RoboDK station: Assembly cell.rdk

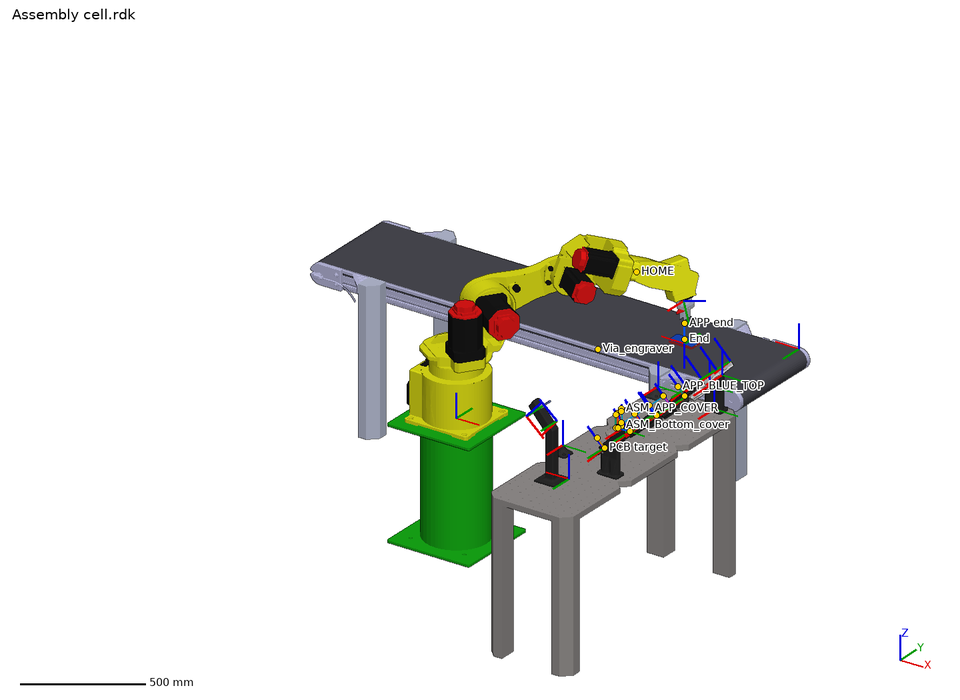
[picture v0: the station drawn from its stored meshes, robots at their saved joint values, targets as dots, program paths as lines]
Station Assembly cell. Poses are relative to the parent item; angles as X-Y-Z fixed-axis rotations.
  - program Assemble Blue phone (11 instructions, listed below)
  - program Assemble Red phone (11 instructions, listed below)
  - folder Frames
    - frame Conveyor Belt Base at (960, 1000, 175) mm, rotated rx 0 ry 0 rz -180 deg
      - robot Conveyor Belt: 1 axes
          modified DH rows (alpha deg, a mm, theta deg, d mm): 0, 0, 0, 0 linear
          base shift (0, 0, 0) mm, rotated rx 0 ry 90 rz 0 deg
          joint limits [-500000] to [500000]; home [0]; saved at [0]
      - frame End distination at (400, 220, 0) mm, rotated rx 180 ry 0 rz 0 deg
        - target End (Cartesian target) at (0, 0, -17.7) mm; joints [55.844, 86.591, -24.189, 14.611, -58.106, -62.758] of M-6IB
        - target APP end  (Cartesian target) at (0, 0, -90) mm; joints [-32.781, 53.881, -40.537, 165.227, 58.581, -48.481] of M-6IB
      - object Ben til Anton samleba at (311, -3, 0) mm, rotated rx -90 ry 0 rz 0 deg, size 80 x 676 x 80 mm, geometry from nd.STEP
      - object Ben til Anton samleba at (1774, -3, 0) mm, rotated rx -90 ry 0 rz -90 deg, size 80 x 676 x 80 mm, geometry from nd.STEP
      - object Ben til Anton samleba at (311, 443, 0) mm, rotated rx -90 ry 0 rz 90 deg, size 80 x 676 x 80 mm, geometry from nd.STEP
      - object Ben til Anton samleba at (1773, 443, 0) mm, rotated rx -90 ry 0 rz 180 deg, size 80 x 676 x 80 mm, geometry from nd.STEP
    - frame M-6IB Base at (0, 0, 0) mm
      - robot M-6IB: 6 axes
          modified DH rows (alpha deg, a mm, theta deg, d mm): 0, 0, 0, 450; -90, 150, -90, 0; 0, 360, 0, 0; -90, 100, 0, 430; 90, 0, 0, 0; -90, 0, 180, 100
          joint limits [-170, -90, -80, -190, -140, -360] to [170, 160, 80, 190, 140, 360]; home [0, 0, 0, 0, 0, 0]; saved at [55.844, 79.928, -20.148, 14.035, -62.022, -61.604]
        - tool TCP_Cover, TCP at (20.4, 0, 95.1) mm, rotated rx 0 ry 15 rz 0 deg
        - tool TCP_DrawingTool(slet mig), TCP at (25.5, 0, 114.13) mm, rotated rx 0 ry 15 rz 0 deg
        - tool TCP_DrawingToolCorner, TCP at (8.96, -4.5, 118.56) mm, rotated rx 180 ry 15 rz 0 deg
        - tool TCP_FUSE, TCP at (19.7, 0, 92.49) mm, rotated rx 0 ry 15 rz 0 deg
        - frame Gripper at (0, 0, 0) mm, rotated rx 90 ry 0 rz -90 deg
          - robot Gripper: 1 axes
              joint limits [0] to [16]; home [0]; saved at [5]
          - target Close (Cartesian target) at (0, 0, 150) mm; joints [0.01] of Gripper
          - target Open (Cartesian target) at (0, 0, 150) mm; joints [5] of Gripper
        - tool TCP_PCB, TCP at (-16.6, 0, 115.3) mm, rotated rx 15 ry 0 rz 90 deg
      - frame Worktable at (700, 400, 175) mm, rotated rx 0 ry 0 rz -90 deg
        - object WorkTable at (20, 20, 0) mm, rotated rx 90 ry 0 rz 0 deg, size 1200 x 700 x 400 mm, geometry from WorkTable.3sections.STEP
        - frame Assembler at (400, 100, 0) mm
          - object Assembler.fixture at (-90, -50, 4) mm, rotated rx -90 ry 0 rz -90 deg, size 70 x 14 x 180 mm, geometry from Assembler.fixture.STEP
          - target ASM_APP_COVER (Cartesian target) at (0, 0, 90) mm, rotated rx -180 ry 0 rz 0 deg; joints [-2.519, 35.979, -52.892, -23.6, -40.23, 111.053] of M-6IB
          - target ASM_APP_FUSE1 (Cartesian target) at (26.19, 0, 80) mm, rotated rx 180 ry 0 rz -90 deg; joints [-2.241, 33.623, -56.565, -1.832, -18.455, 3.903] of M-6IB
          - target ASM_APP_FUSE2 (Cartesian target) at (39.25, 0, 80) mm, rotated rx 180 ry 0 rz -90 deg; joints [-3.357, 33.698, -56.518, -2.734, -18.526, 5.835] of M-6IB
          - target ASM_APP_PCB (Cartesian target) at (0, 0, 80) mm, rotated rx 180 ry 0 rz -180 deg; joints [2.519, 37.294, -54.217, 24.249, -39.018, -111.896] of M-6IB
          - target ASM_Bottom_cover (Cartesian target) at (0, 0, 17) mm, rotated rx 180 ry 0 rz 0 deg; joints [-2.519, 44.305, -60.421, -27.98, -33.444, -243.485] of M-6IB
          - target ASM_FUSE1 (Cartesian target) at (26.19, 0, 19.5) mm, rotated rx 180 ry 0 rz -90 deg; joints [-2.241, 40.726, -62.911, -2.764, -12.114, 4.868] of M-6IB
          - target ASM_FUSE2 (Cartesian target) at (39.25, 0, 19.5) mm, rotated rx 180 ry 0 rz -90 deg; joints [-3.357, 40.792, -62.856, -4.112, -12.199, 7.262] of M-6IB
          - target ASM_GRAB_PHONE (Cartesian target) at (0, 0, 23.7) mm, rotated rx -180 ry 0 rz 0 deg; joints [-2.519, 43.211, -59.538, -27.369, -34.225, 115.779] of M-6IB
          - target ASM_PCB (Cartesian target) at (0, 0, 14.5) mm, rotated rx 180 ry 0 rz 180 deg; joints [0, 25.65, -72.841, 0, -2.159, 0] of M-6IB
          - target ASM_TOP_cover (Cartesian target) at (0, 0, 28.7) mm, rotated rx 180 ry 0 rz 0 deg; joints [-2.519, 42.635, -59.062, -27.052, -34.649, 115.394] of M-6IB
          - object Assembler.fixture at (-90, -50, 4) mm, rotated rx -90 ry 0 rz -90 deg, size 70 x 14 x 180 mm, geometry from Assembler.fixture.STEP
          - target HOME (Cartesian target) at (0, 75.1, 714.6) mm, rotated rx -180 ry 75 rz -90 deg; joints [0, 0, 0, 0, 0, 0] of M-6IB
          - object Sikring at (-790, -279.25, 13.5) mm, rotated rx 0 ry -45 rz -90 deg, size 5 x 20 x 5 mm, geometry from Sikring.STEP
          - object Sikring at (-790, -266.19, 13.5) mm, rotated rx 0 ry -45 rz -90 deg, size 5 x 20 x 5 mm, geometry from Sikring.STEP
          - object PCB at (-780, -245.3, 6.2) mm, rotated rx -90 ry 0 rz 0 deg, size 55 x 11.2 x 106.7 mm, geometry from PCB.STEP
          - object BundRed at (-780, -240, 11) mm, rotated rx 0 ry 0 rz -90 deg, size 60 x 13 x 114 mm, geometry from BundRed.STEP
          - object TopBlue at (-780, -240, 17.7) mm, rotated rx 0 ry 0 rz -90 deg, size 60 x 11.7 x 114 mm, geometry from TopBlue.STEP
        - frame Calibration tip 2 at (720, 40, 40) mm
          - object Calibration tip2 - Table at (0, 0, -40) mm, rotated rx 90 ry 0 rz 0 deg, size 64 x 40 x 64 mm, geometry from Calibration tip - Table.STEP
        - frame Engraving tool at (890, 190, 0) mm, rotated rx 0 ry 0 rz -90 deg
          - frame Pencil at (171.86, 50, 249.32) mm, rotated rx 0 ry 41.29 rz -180 deg
            - target Via_engraver (Cartesian target) at (-59.9, 461.47, 104.18) mm, rotated rx -165.52 ry -18.84 rz -114.89 deg; joints [-18.02, 30.15, -78.63, -152.85, -139.18, 114.67] of M-6IB
          - frame Pencil corner(slet mig) at (31.87, 41, 263.19) mm, rotated rx 0 ry 48.71 rz 0 deg
          - object Engraving Tool at (0, 0, 0) mm, rotated rx -90 ry 0 rz 0 deg, size 171.9 x 351.3 x 100 mm, geometry from Pencil.assembly.STEP
        - frame Left Pillar at (40, 300, 0) mm
          - frame Rod lower at (-11.02, -32.53, 91.11) mm
            - object Rod at (0, 0, 0) mm, size 8 x 742 x 8 mm, geometry from Rod.STEP
            - frame Assembly blue bottom cover 1 at (250, 137.68, 167.7) mm, rotated rx 0 ry 45 rz -90 deg
              - frame target_blue_bottom_cover at (280, 35.13, -4.5) mm
                - target Blue_bottom (Cartesian target) at (0, 0, 0) mm, rotated rx 180 ry 0 rz 0 deg; joints [7.51, 44.296, -67.681, -10.607, 37.945, 4.63] of M-6IB
                - target APP_Blue_bottom (Cartesian target) at (0, 0, 50) mm, rotated rx 180 ry 0 rz 0 deg; joints [7.935, 36.225, -67.101, -11.351, 37.406, 5.073] of M-6IB
                - object BundBlue at (0, 0, 0) mm, size 60 x 13 x 114 mm, geometry from BundBlue.STEP
              - object Top cover fixture at (0, 0, 0) mm, size 70.2 x 39.6 x 342 mm, geometry from Top cover fixture.STEP
              - object FixtureBlack at (0, 0, 1.25) mm, rotated rx 0 ry 0 rz 180 deg, size 342 x 70.2 x 41.2 mm, geometry from FixtureBlack.STEP
            - frame Assembly blue top cover 1 at (50, 137.68, 167.7) mm, rotated rx 0 ry 45 rz -90 deg
              - frame target_blue_top_cover at (280, 35.12, -4.5) mm
                - target BLUE_TOP (Cartesian target) at (0, 0, 5) mm, rotated rx 180 ry 0 rz 0 deg; joints [23.805, 48.879, -62.525, -36.506, 35.985, 18.478] of M-6IB
                - target APP_BLUE_TOP (Cartesian target) at (0, 0, 50) mm, rotated rx 180 ry 0 rz 0 deg; joints [24.889, 42.011, -62.308, -38.195, 36.117, 19.379] of M-6IB
              - object Top cover fixture at (0, 0, 0) mm, size 70.2 x 39.6 x 342 mm, geometry from Top cover fixture.STEP
            - frame Assembly red bottom cover 2 at (350, 137.68, 167.7) mm, rotated rx 0 ry 45 rz -90 deg
              - frame target_red_bottom_cover at (280, 35.12, -4.5) mm
                - target Red_bottom (Cartesian target) at (0, 0, 0) mm, rotated rx 180 ry 0 rz 0 deg; joints [-1.236, 44.216, -68.191, 181.732, -38.198, -180.743] of M-6IB
                - target APP_Red_bottom (Cartesian target) at (0, 0, 50) mm, rotated rx 180 ry 0 rz 0 deg; joints [-1.307, 36.105, -67.625, 181.854, -37.633, -180.815] of M-6IB
              - object FixtureBlack at (0, 0, 1.25) mm, rotated rx 0 ry 0 rz 180 deg, size 342 x 70.2 x 41.2 mm, geometry from FixtureBlack.STEP
            - frame Assembly red top cover 2 at (150, 137.68, 167.7) mm, rotated rx 0 ry 45 rz -90 deg
              - object Top cover fixture at (0, 0, 0) mm, size 70.2 x 39.6 x 342 mm, geometry from Top cover fixture.STEP
              - frame target_red_top_cover at (280, 35.12, -4.5) mm
                - target Red_top (Cartesian target) at (0, 0, 5) mm, rotated rx 180 ry 0 rz 0 deg; joints [16.006, 45.457, -65.78, -23.315, 37.109, 10.806] of M-6IB
                - target APP_Red_top (Cartesian target) at (0, 0, 50) mm, rotated rx 180 ry 0 rz 0 deg; joints [16.787, 38.357, -65.346, -24.653, 36.843, 11.591] of M-6IB
                - object TopRed at (0, 0, 0) mm, size 60 x 11.7 x 114 mm, geometry from TopRed.STEP
              - object Top cover fixture at (0, 0, 0) mm, size 70.2 x 39.6 x 342 mm, geometry from Top cover fixture.STEP
            - frame Fuses fixture at (500, 83.09, 94.4) mm, rotated rx 0 ry 45 rz -90 deg
              - frame fuse target at (154.59, 6.25, 7) mm
                - target Fuse target (Cartesian target) at (0, 0, 0) mm, rotated rx 135 ry 0 rz -90 deg; joints [-10.843, 50.524, -86.333, -184.166, -86.343, 90.266] of M-6IB
                - target APP_Target_fuse (Cartesian target) at (40, 0, 40) mm, rotated rx 180 ry 0 rz -90 deg; joints [-9.229, 37.854, -63.685, -23.305, 21.644, -61.596] of M-6IB
                - object Sikring at (0, -10, 0) mm, size 5 x 20 x 5 mm, geometry from Sikring.STEP
                - object Sikring at (0, -10, 0) mm, size 5 x 20 x 5 mm, geometry from Sikring.STEP
              - object FuseFixture at (0, 0, 0) mm, size 28.5 x 33.2 x 160 mm, geometry from FuseFixture.STEP
            - frame PCB fixture at (600, 90.16, 101.47) mm, rotated rx 0 ry 45 rz -90 deg
              - frame pcb target at (187.5, 64.5, 6.5) mm
                - target PCB target (Cartesian target) at (0, -5.3, 0) mm, rotated rx 180 ry 0 rz -90 deg; joints [-28.731, 41.343, -74.438, -145.13, -46.732, -190.202] of M-6IB
                - target APP_PCB (Cartesian target) at (0, -5.3, 50) mm, rotated rx 180 ry 0 rz -90 deg; joints [0, 0, 0, 0, 0, 0] of M-6IB
              - object PCB fixture at (0, 0, 0) mm, rotated rx 90 ry 0 rz 90 deg, size 118 x 39.5 x 220 mm, geometry from PCB fixture.STEP
          - frame Rod upper at (-11.02, 31.11, 154.75) mm
            - object Rod at (0, 0, 0) mm, size 8 x 742 x 8 mm, geometry from Rod.STEP
          - object Pillar at (0, 0, 0) mm, rotated rx 90 ry 0 rz 0 deg, size 60 x 165 x 100 mm, geometry from Søjle.STEP
        - frame Right Pillar at (760, 300, 0) mm
          - object Pillar at (0, 0, 0) mm, rotated rx 90 ry 0 rz 0 deg, size 60 x 165 x 100 mm, geometry from Søjle.STEP
        - frame Calibration tip 1 at (80, 40, 40) mm
          - object Calibration tip - Table at (0, 0, -40) mm, rotated rx 90 ry 0 rz 0 deg, size 64 x 40 x 64 mm, geometry from Calibration tip - Table.STEP
  - folder Programs
    - folder Attach Programs
      - program Attach_Bottom_Cover_Blue (8 instructions, listed below)
      - program Attach_Bottom_Cover_Red (8 instructions, listed below)
      - program Attach_Top_Cover_Blue (8 instructions, listed below)
      - program Attach_Top_Cover_Red (8 instructions, listed below)
      - program Attach_PCB (8 instructions, listed below)
      - program Attach_phone (10 instructions, listed below)
      - program Attach_Fuse (8 instructions, listed below)
    - folder Detach Programs
      - program Detach_Fuse1 (6 instructions, listed below)
      - program Detach_Fuse2 (6 instructions, listed below)
      - program Detach_PCB (7 instructions, listed below)
      - program Detach_Bottom (6 instructions, listed below)
      - program Detach_Top (5 instructions, listed below)
    - folder Misc
      - frame Robotbase_frame at (0, 0, -525) mm
        - object RobotBase at (-200, -200, 0) mm, rotated rx 90 ry 0 rz 0 deg, size 400 x 525 x 400 mm, geometry from RobotBase.STEP
      - program Open gripper (4 instructions, listed below)
      - program Close gripper (1 instructions, listed below)
      - Python program Generate G-Code (listed below)
      - Python program Import G-Code (listed below)
      - program Final step (6 instructions, listed below)
    - program Reset 2 (1 instructions, listed below)
    - folder Programs for Test
      - program Red phone assembly test (2 instructions, listed below)
      - program Blue phone assembly test (2 instructions, listed below)
  - Python program Assemble red phone (listed below)
  - program Reset (2 instructions, listed below)
  - Python program Assemble blue phone (listed below)
  - program AssembleInterior (6 instructions, listed below)
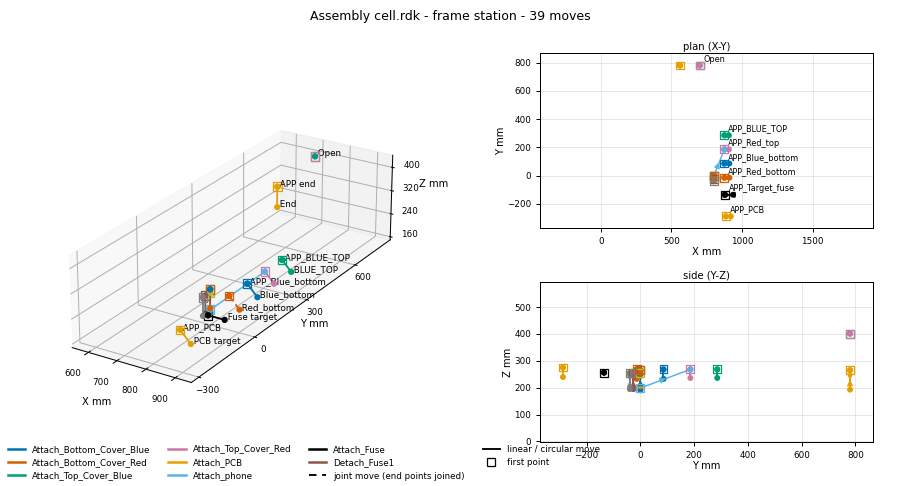
[picture p0: tool path of Assembly cell.rdk in frame station, 39 of 39 moves have a stored position in this frame; points joined in program order, loops and branches not executed]

--- program Assemble Blue phone (robot M-6IB) ---
  Call Attach_Bottom_Cover_Blue
  Call Detach_Bottom
  Call Attach_PCB
  Call Detach_PCB
  Call Attach_Fuse
  Call Detach_Fuse1
  Call Attach_Fuse
  Call Detach_Fuse2
  Call Attach_Top_Cover_Blue
  Call Detach_Top
  Call Final step

--- program Assemble Red phone (robot M-6IB) ---
  Call Attach_Bottom_Cover_Red
  Call Detach_Bottom
  Call Attach_PCB
  Call Detach_PCB
  Call Attach_Fuse
  Call Detach_Fuse1
  Call Attach_Fuse
  Call Detach_Fuse2
  Call Attach_Top_Cover_Red
  Call Detach_Top
  Call Final step

--- program Attach_Bottom_Cover_Blue (robot M-6IB) ---
  Set Tool: TCP_Cover
  Set Ref.: target_blue_bottom_cover
  Call Open
  MoveJ (APP_Blue_bottom)
  MoveL (Blue_bottom)
  Attach to TCP_PCB
  Call Close gripper
  MoveL (APP_Blue_bottom)

--- program Attach_Bottom_Cover_Red (robot M-6IB) ---
  Set Tool: TCP_Cover
  Set Ref.: target_red_bottom_cover
  Call Open
  MoveJ (APP_Red_bottom)
  MoveJ (Red_bottom)
  Attach to TCP_PCB
  Call Close gripper
  MoveJ (APP_Red_bottom)

--- program Attach_Top_Cover_Blue (robot M-6IB) ---
  Set Tool: TCP_Cover
  Set Ref.: target_blue_top_cover
  Call Open
  MoveJ (APP_BLUE_TOP)
  MoveL (BLUE_TOP)
  Attach to TCP_PCB
  Call Close gripper
  MoveL (APP_BLUE_TOP)

--- program Attach_Top_Cover_Red (robot M-6IB) ---
  Set Tool: TCP_Cover
  Set Ref.: target_red_top_cover
  Call Open
  MoveJ (APP_Red_top)
  MoveL (Red_top)
  Attach to TCP_PCB
  Call Close gripper
  MoveL (APP_Red_top)

--- program Attach_PCB (robot M-6IB) ---
  Set Tool: TCP_PCB
  Set Ref.: pcb target
  Call Open
  MoveJ (APP_PCB)
  MoveL (PCB target)
  Attach to TCP_PCB
  Call Close gripper
  MoveL (APP_PCB)

--- program Attach_phone (robot M-6IB) ---
  Set Tool: TCP_Cover
  Set Ref.: Assembler
  MoveL (ASM_GRAB_PHONE)
  Call Close gripper
  Attach to TCP_Cover
  Attach to TCP_Cover
  Attach to TCP_Cover
  Attach to TCP_Cover
  Attach to TCP_Cover
  MoveL (APP_Red_top)

--- program Attach_Fuse (robot M-6IB) ---
  Set Tool: TCP_FUSE
  Set Ref.: fuse target
  Call Open
  MoveJ (APP_Target_fuse)
  MoveL (Fuse target)
  Attach to TCP_PCB
  Call Close gripper
  MoveL (APP_Target_fuse)

--- program Detach_Fuse1 (robot M-6IB) ---
  Set Ref.: Assembler
  Set Tool: TCP_FUSE
  MoveJ (ASM_APP_FUSE1)
  MoveL (ASM_FUSE1)
  Call Open gripper
  MoveL (ASM_APP_FUSE1)

--- program Detach_Fuse2 (robot M-6IB) ---
  Set Ref.: Assembler
  Set Tool: TCP_FUSE
  MoveJ (ASM_APP_FUSE2)
  MoveL (ASM_FUSE2)
  Call Open gripper
  MoveL (ASM_APP_FUSE2)

--- program Detach_PCB (robot M-6IB) ---
  Set Ref.: Assembler
  Set Tool: TCP_PCB
  MoveJ (ASM_APP_PCB)
  MoveL (ASM_PCB)
  Call Open gripper
  Replace PCB
  MoveL (ASM_APP_PCB)

--- program Detach_Bottom (robot M-6IB) ---
  Set Ref.: Assembler
  Set Tool: TCP_Cover
  MoveJ (ASM_APP_COVER)
  MoveL (ASM_Bottom_cover)
  Call Open gripper
  MoveL (ASM_APP_COVER)

--- program Detach_Top (robot M-6IB) ---
  Set Ref.: Assembler
  Set Tool: TCP_Cover
  MoveJ (ASM_APP_COVER)
  MoveL (ASM_TOP_cover)
  Call Open gripper

--- program Open gripper (robot Gripper) ---
  MoveJ (Open)
  Detach from TCP_Cover
  Detach from TCP_PCB
  Detach from TCP_FUSE

--- program Close gripper (robot Gripper) ---
  MoveJ (Close)

--- Python program Generate G-Code ---
# Typo created by Adrien Rosselet

from os import path               # Operating System API
from robolink import *    # RoboDK API
from robodk import *      # Robot toolbox
#import time
import sys                # System specific
#Connect to RoboDK
RDK = Robolink()

#If no input the text equals ROBOT.
text = 'ROBOT'
#Use function call argument as text.
if len(sys.argv) > 1:
    text = sys.argv[1]

#Set file directory for G-code file
filedirectory = path.expandvars(r'%USERPROFILE%\AppData\Local\Temp\letters.gcode')

# parametres (in mm)
lengthLet = 6  # minimum half of hightLet
hightLet = 9  # letter hight
space = 2  # space between letters
depth = 0.3  # engraving depth
up = -3  # hight when the tool is mooving
fileID = open(filedirectory, 'w')  # enter the name of the created fileID
# Header line for G-code
fileID.write(str(('%s\n' % 'G21 G90 G17 F1500')))

# program
down = depth
posAct = 0  # X value of actual position

#G-code parameters
fileID.write(str(('%s\n' % 'G01 X0 Y0 Z1')))
rapide = 'G0'
lent = 'G01'
tourHoraire = 'G02'
tourAntihoraire = 'G03'
total_lenght = len(text)*lengthLet




for elem in text:
    if elem == 'A':
            fileID.write(str(('%s %c%f %c%f %c%f\n' % (
                              rapide, 'X', posAct, 'Y', 0, 'Z', up))))
            fileID.write(str(('%s %c%f %c%f %c%f\n' % (
                         lent, 'X', posAct, 'Y', 0, 'Z', down))))
            fileID.write(str(('%s %c%f %c%f %c%f\n' % ( lent, 'X',
                         posAct+lengthLet/2, 'Y', hightLet, 'Z', down))))
            fileID.write(str(('%s %c%f %c%f %c%f\n' % ( lent,
                         'X', posAct+lengthLet, 'Y', 0, 'Z', down))))
            fileID.write(str(('%s %c%f %c%f %c%f\n' % ( rapide,
                         'X', posAct+lengthLet, 'Y', 0, 'Z', up))))
            fileID.write(str(('%s %c%f %c%f %c%f\n' % ( rapide, 'X',
                         posAct+lengthLet/4, 'Y', hightLet/2, 'Z', up))))
            fileID.write(str(('%s %c%f %c%f %c%f\n' % ( lent, 'X',
                         posAct+lengthLet/4, 'Y', hightLet/2, 'Z', down))))
            fileID.write(str(('%s %c%f %c%f %c%f\n' % ( lent, 'X',
                         posAct+lengthLet*3/4, 'Y', hightLet/2, 'Z', down))))
            fileID.write(str(('%s %c%f %c%f %c%f\n' % ( rapide, 'X',
                         posAct+lengthLet*3/4, 'Y', hightLet/2, 'Z', up))))
            posAct = posAct+lengthLet
    elif elem == 'B':
            fileID.write(str(('%s %c%f %c%f %c%f\n' % (
                         rapide, 'X', posAct, 'Y', 0, 'Z', up))))
            fileID.write(str(('%s %c%f %c%f %c%f\n' % (
                         lent, 'X', posAct, 'Y', 0, 'Z', down))))
            fileID.write(str(('%s %c%f %c%f %c%f\n' % ( lent,
                         'X', posAct, 'Y', hightLet, 'Z', down))))
            fileID.write(str(('%s %c%f %c%f %c%f\n' % ( lent, 'X',
                         posAct+lengthLet-hightLet/4, 'Y', hightLet, 'Z', down))))
            fileID.write(str(('%s %c%f %c%f %c%f %c%f\n' % ( tourHoraire, 'X',
                         posAct+lengthLet-hightLet/4, 'Y', hightLet/2, 'I', 0, 'J', -hightLet/4))))
            fileID.write(str(('%s %c%f %c%f %c%f\n' % ( lent,
                         'X', posAct, 'Y', hightLet/2, 'Z', down))))
            fileID.write(str(('%s %c%f %c%f %c%f\n' % ( lent, 'X',
                         posAct+lengthLet-hightLet/4, 'Y', hightLet/2, 'Z', down))))
            fileID.write(str(('%s %c%f %c%f %c%f %c%f\n' % ( tourHoraire, 'X',
                         posAct+lengthLet-hightLet/4, 'Y', 0, 'I', 0, 'J', -hightLet/4))))
            fileID.write(str(('%s %c%f %c%f %c%f\n' % (
                         lent, 'X', posAct, 'Y', 0, 'Z', down))))
            fileID.write(str(('%s %c%f %c%f %c%f\n' % (
                         rapide, 'X', posAct, 'Y', 0, 'Z', up))))
            posAct = posAct+lengthLet
    elif elem == 'C':
            fileID.write(str(('%s %c%f %c%f %c%f\n' % ( rapide, 'X',
                         posAct+lengthLet, 'Y', hightLet*3/4, 'Z', up))))
            fileID.write(str(('%s %c%f %c%f %c%f\n' % ( lent, 'X',
                         posAct+lengthLet, 'Y', hightLet*3/4, 'Z', down))))
            fileID.write(str(('%s %c%f %c%f %c%f %c%f\n' % ( tourAntihoraire, 'X',
                         posAct+lengthLet-hightLet/4, 'Y', hightLet, 'I', -hightLet/4, 'J', 0))))
            fileID.write(str(('%s %c%f %c%f %c%f\n' % ( lent, 'X',
                         posAct+hightLet/4, 'Y', hightLet, 'Z', down))))
            fileID.write(str(('%s %c%f %c%f %c%f %c%f\n' % ( tourAntihoraire,
                         'X', posAct, 'Y', hightLet*3/4, 'I', 0, 'J', -hightLet/4))))
            fileID.write(str(('%s %c%f %c%f %c%f\n' % ( lent,
                         'X', posAct, 'Y', hightLet/4, 'Z', down))))
            fileID.write(str(('%s %c%f %c%f %c%f %c%f\n' % ( tourAntihoraire,
                         'X', posAct+hightLet/4, 'Y', 0, 'I', hightLet/4, 'J', 0))))
            fileID.write(str(('%s %c%f %c%f %c%f\n' % ( lent, 'X',
                         posAct+lengthLet-hightLet/4, 'Y', 0, 'Z', down))))
            fileID.write(str(('%s %c%f %c%f %c%f %c%f\n' % ( tourAntihoraire,
                         'X', posAct+lengthLet, 'Y', hightLet/4, 'I', 0, 'J', hightLet/4))))
            fileID.write(str(('%s %c%f %c%f %c%f\n' % ( rapide,
                         'X', posAct+lengthLet, 'Y', hightLet/4, 'Z', up))))
            posAct = posAct+lengthLet
    elif elem == 'D':
            fileID.write(str(('%s %c%f %c%f %c%f\n' % (
                         rapide, 'X', posAct, 'Y', 0, 'Z', up))))
            fileID.write(str(('%s %c%f %c%f %c%f\n' % (
                         lent, 'X', posAct, 'Y', 0, 'Z', down))))
            fileID.write(str(('%s %c%f %c%f %c%f\n' % ( lent,
                         'X', posAct, 'Y', hightLet, 'Z', down))))
            fileID.write(str(('%s %c%f %c%f %c%f\n' % ( lent, 'X',
                         posAct+lengthLet-hightLet/2, 'Y', hightLet, 'Z', down))))
            fileID.write(str(('%s %c%f %c%f %c%f %c%f\n' % ( tourHoraire, 'X',
                         posAct+lengthLet-hightLet/2, 'Y', 0, 'I', 0, 'J', -hightLet/2))))
            fileID.write(str(('%s %c%f %c%f %c%f\n' % (
                         lent, 'X', posAct, 'Y', 0, 'Z', down))))
            fileID.write(str(('%s %c%f %c%f %c%f\n' % (
                         rapide, 'X', posAct, 'Y', 0, 'Z', up))))
            posAct = posAct+lengthLet
    elif elem == 'E':
            fileID.write(str(('%s %c%f %c%f %c%f\n' % (
                         rapide, 'X', posAct, 'Y', 0, 'Z', up))))
            fileID.write(str(('%s %c%f %c%f %c%f\n' % (
                         lent, 'X', posAct, 'Y', 0, 'Z', down))))
            fileID.write(str(('%s %c%f %c%f %c%f\n' % ( lent,
                         'X', posAct, 'Y', hightLet, 'Z', down))))
            fileID.write(str(('%s %c%f %c%f %c%f\n' % ( lent, 'X',
                         posAct+lengthLet, 'Y', hightLet, 'Z', down))))
            fileID.write(str(('%s %c%f %c%f %c%f\n' % ( rapide,
                         'X', posAct+lengthLet, 'Y', hightLet, 'Z', up))))
            fileID.write(str(('%s %c%f %c%f %c%f\n' % ( rapide,
                         'X', posAct, 'Y', hightLet/2, 'Z', up))))
            fileID.write(str(('%s %c%f %c%f %c%f\n' % ( lent,
                         'X', posAct, 'Y', hightLet/2, 'Z', down))))
            fileID.write(str(('%s %c%f %c%f %c%f\n' % ( lent, 'X',
                         posAct+lengthLet, 'Y', hightLet/2, 'Z', down))))
            fileID.write(str(('%s %c%f %c%f %c%f\n' % ( rapide,
                         'X', posAct+lengthLet, 'Y', hightLet/2, 'Z', up))))
            fileID.write(str(('%s %c%f %c%f %c%f\n' % (
                         rapide, 'X', posAct, 'Y', 0, 'Z', up))))
            fileID.write(str(('%s %c%f %c%f %c%f\n' % (
                         lent, 'X', posAct, 'Y', 0, 'Z', down))))
            fileID.write(str(('%s %c%f %c%f %c%f\n' % ( lent,
                         'X', posAct+lengthLet, 'Y', 0, 'Z', down))))
            fileID.write(str(('%s %c%f %c%f %c%f\n' % ( rapide,
                         'X', posAct+lengthLet, 'Y', 0, 'Z', up))))
            posAct = posAct+lengthLet
    elif elem == 'F':
            fileID.write(str(('%s %c%f %c%f %c%f\n' % (
                         rapide, 'X', posAct, 'Y', 0, 'Z', up))))
            fileID.write(str(('%s %c%f %c%f %c%f\n' % (
                         lent, 'X', posAct, 'Y', 0, 'Z', down))))
            fileID.write(str(('%s %c%f %c%f %c%f\n' % ( lent,
                         'X', posAct, 'Y', hightLet, 'Z', down))))
            fileID.write(str(('%s %c%f %c%f %c%f\n' % ( lent, 'X',
                         posAct+lengthLet, 'Y', hightLet, 'Z', down))))
            fileID.write(str(('%s %c%f %c%f %c%f\n' % ( rapide,
                         'X', posAct+lengthLet, 'Y', hightLet, 'Z', up))))
            fileID.write(str(('%s %c%f %c%f %c%f\n' % ( rapide,
                         'X', posAct, 'Y', hightLet/2, 'Z', up))))
            fileID.write(str(('%s %c%f %c%f %c%f\n' % ( lent,
                         'X', posAct, 'Y', hightLet/2, 'Z', down))))
            fileID.write(str(('%s %c%f %c%f %c%f\n' % ( lent, 'X',
                         posAct+lengthLet, 'Y', hightLet/2, 'Z', down))))
            fileID.write(str(('%s %c%f %c%f %c%f\n' % ( rapide,
                         'X', posAct+lengthLet, 'Y', hightLet/2, 'Z', up))))
            posAct = posAct+lengthLet
    elif elem == 'G':
            fileID.write(str(('%s %c%f %c%f %c%f\n' % ( rapide, 'X',
                         posAct+lengthLet, 'Y', hightLet*3/4, 'Z', up))))
            fileID.write(str(('%s %c%f %c%f %c%f\n' % ( lent, 'X',
                         posAct+lengthLet, 'Y', hightLet*3/4, 'Z', down))))
            fileID.write(str(('%s %c%f %c%f %c%f %c%f\n' % ( tourAntihoraire, 'X',
                         posAct+lengthLet-hightLet/4, 'Y', hightLet, 'I', -hightLet/4, 'J', 0))))
            fileID.write(str(('%s %c%f %c%f %c%f\n' % ( lent, 'X',
                         posAct+hightLet/4, 'Y', hightLet, 'Z', down))))
            fileID.write(str(('%s %c%f %c%f %c%f %c%f\n' % ( tourAntihoraire,
                         'X', posAct, 'Y', hightLet*3/4, 'I', 0, 'J', -hightLet/4))))
            fileID.write(str(('%s %c%f %c%f %c%f\n' % ( lent,
                         'X', posAct, 'Y', hightLet/4, 'Z', down))))
            fileID.write(str(('%s %c%f %c%f %c%f %c%f\n' % ( tourAntihoraire,
                         'X', posAct+hightLet/4, 'Y', 0, 'I', hightLet/4, 'J', 0))))
            fileID.write(str(('%s %c%f %c%f %c%f\n' % ( lent, 'X',
                         posAct+lengthLet-hightLet/4, 'Y', 0, 'Z', down))))
            fileID.write(str(('%s %c%f %c%f %c%f %c%f\n' % ( tourAntihoraire,
                         'X', posAct+lengthLet, 'Y', hightLet/4, 'I', 0, 'J', hightLet/4))))
            fileID.write(str(('%s %c%f %c%f %c%f\n' % ( lent, 'X',
                         posAct+lengthLet, 'Y', hightLet/2, 'Z', down))))
            fileID.write(str(('%s %c%f %c%f %c%f\n' % ( lent, 'X',
                         posAct+lengthLet/2, 'Y', hightLet/2, 'Z', down))))
            fileID.write(str(('%s %c%f %c%f %c%f\n' % ( rapide, 'X',
                         posAct+lengthLet/2, 'Y', hightLet/2, 'Z', up))))
            posAct = posAct+lengthLet
    elif elem == 'H':
            fileID.write(str(('%s %c%f %c%f %c%f\n' % (
                         rapide, 'X', posAct, 'Y', 0, 'Z', up))))
            fileID.write(str(('%s %c%f %c%f %c%f\n' % (
                         lent, 'X', posAct, 'Y', 0, 'Z', down))))
            fileID.write(str(('%s %c%f %c%f %c%f\n' % ( lent,
                         'X', posAct, 'Y', hightLet, 'Z', down))))
            fileID.write(str(('%s %c%f %c%f %c%f\n' % (
                         rapide, 'X', posAct, 'Y', hightLet, 'Z', up))))
            fileID.write(str(('%s %c%f %c%f %c%f\n' % ( rapide,
                         'X', posAct+lengthLet, 'Y', 0, 'Z', up))))
            fileID.write(str(('%s %c%f %c%f %c%f\n' % ( lent,
                         'X', posAct+lengthLet, 'Y', 0, 'Z', down))))
            fileID.write(str(('%s %c%f %c%f %c%f\n' % ( lent, 'X',
                         posAct+lengthLet, 'Y', hightLet, 'Z', down))))
            fileID.write(str(('%s %c%f %c%f %c%f\n' % ( rapide,
                         'X', posAct+lengthLet, 'Y', hightLet, 'Z', up))))
            fileID.write(str(('%s %c%f %c%f %c%f\n' % ( rapide,
                         'X', posAct, 'Y', hightLet/2, 'Z', up))))
            fileID.write(str(('%s %c%f %c%f %c%f\n' % ( lent,
                         'X', posAct, 'Y', hightLet/2, 'Z', down))))
            fileID.write(str(('%s %c%f %c%f %c%f\n' % ( lent, 'X',
                         posAct+lengthLet, 'Y', hightLet/2, 'Z', down))))
            fileID.write(str(('%s %c%f %c%f %c%f\n' % ( rapide,
                         'X', posAct+lengthLet, 'Y', hightLet/2, 'Z', up))))
            posAct = posAct+lengthLet
    elif elem == 'I':
            fileID.write(str(('%s %c%f %c%f %c%f\n' % ( rapide,
                         'X', posAct+lengthLet/4, 'Y', 0, 'Z', up))))
            fileID.write(str(('%s %c%f %c%f %c%f\n' % ( lent,
                         'X', posAct+lengthLet/4, 'Y', 0, 'Z', down))))
            fileID.write(str(('%s %c%f %c%f %c%f\n' % ( lent, 'X',
                         posAct+lengthLet/4, 'Y', hightLet, 'Z', down))))
            fileID.write(str(('%s %c%f %c%f %c%f\n' % ( rapide,
                         'X', posAct+lengthLet/4, 'Y', hightLet, 'Z', up))))
            fileID.write(str(('%s %c%f %c%f %c%f\n' % (
                         rapide, 'X', posAct, 'Y', hightLet, 'Z', up))))
            fileID.write(str(('%s %c%f %c%f %c%f\n' % ( lent,
                         'X', posAct, 'Y', hightLet, 'Z', down))))
            fileID.write(str(('%s %c%f %c%f %c%f\n' % ( lent, 'X',
                         posAct+lengthLet/2, 'Y', hightLet, 'Z', down))))
            fileID.write(str(('%s %c%f %c%f %c%f\n' % ( rapide,
                         'X', posAct+lengthLet/2, 'Y', hightLet, 'Z', up))))
            fileID.write(str(('%s %c%f %c%f %c%f\n' % (
                         rapide, 'X', posAct, 'Y', 0, 'Z', up))))
            fileID.write(str(('%s %c%f %c%f %c%f\n' % (
                         lent, 'X', posAct, 'Y', 0, 'Z', down))))
            fileID.write(str(('%s %c%f %c%f %c%f\n' % ( lent,
                         'X', posAct+lengthLet/2, 'Y', 0, 'Z', down))))
            fileID.write(str(('%s %c%f %c%f %c%f\n' % ( rapide,
                         'X', posAct+lengthLet/2, 'Y', 0, 'Z', up))))
            posAct = posAct+lengthLet/2
    elif elem == 'J':
            fileID.write(str(('%s %c%f %c%f %c%f\n' % ( rapide,
                         'X', posAct, 'Y', hightLet/4, 'Z', up))))
            fileID.write(str(('%s %c%f %c%f %c%f\n' % ( lent,
                         'X', posAct, 'Y', hightLet/4, 'Z', down))))
            fileID.write(str(('%s %c%f %c%f %c%f %c%f\n' % ( tourAntihoraire,
                         'X', posAct+hightLet/4, 'Y', 0, 'I', +hightLet/4, 'J', 0))))
            fileID.write(str(('%s %c%f %c%f %c%f\n' % ( lent, 'X',
                         posAct+lengthLet-hightLet/4, 'Y', 0, 'Z', down))))
            fileID.write(str(('%s %c%f %c%f %c%f %c%f\n' % ( tourAntihoraire,
                         'X', posAct+lengthLet, 'Y', hightLet/4, 'I', 0, 'J', +hightLet/4))))
            fileID.write(str(('%s %c%f %c%f %c%f\n' % ( lent, 'X',
                         posAct+lengthLet, 'Y', hightLet, 'Z', down))))
            fileID.write(str(('%s %c%f %c%f %c%f\n' % ( lent,
                         'X', posAct, 'Y', hightLet, 'Z', down))))
            fileID.write(str(('%s %c%f %c%f %c%f\n' % (
                         rapide, 'X', posAct, 'Y', hightLet, 'Z', up))))
            posAct = posAct+lengthLet
    elif elem == 'K':
            fileID.write(str(('%s %c%f %c%f %c%f\n' % (
                         rapide, 'X', posAct, 'Y', 0, 'Z', up))))
            fileID.write(str(('%s %c%f %c%f %c%f\n' % (
                         lent, 'X', posAct, 'Y', 0, 'Z', down))))
            fileID.write(str(('%s %c%f %c%f %c%f\n' % ( lent,
                         'X', posAct, 'Y', hightLet, 'Z', down))))
            fileID.write(str(('%s %c%f %c%f %c%f\n' % (
                         rapide, 'X', posAct, 'Y', hightLet, 'Z', up))))
            fileID.write(str(('%s %c%f %c%f %c%f\n' % ( rapide,
                         'X', posAct, 'Y', hightLet/2, 'Z', up))))
            fileID.write(str(('%s %c%f %c%f %c%f\n' % ( lent,
                         'X', posAct, 'Y', hightLet/2, 'Z', down))))
            fileID.write(str(('%s %c%f %c%f %c%f\n' % ( lent, 'X',
                         posAct+lengthLet, 'Y', hightLet, 'Z', down))))
            fileID.write(str(('%s %c%f %c%f %c%f\n' % ( rapide,
                         'X', posAct+lengthLet, 'Y', hightLet, 'Z', up))))
            fileID.write(str(('%s %c%f %c%f %c%f\n' % ( rapide,
                         'X', posAct, 'Y', hightLet/2, 'Z', up))))
            fileID.write(str(('%s %c%f %c%f %c%f\n' % ( lent,
                         'X', posAct, 'Y', hightLet/2, 'Z', down))))
            fileID.write(str(('%s %c%f %c%f %c%f\n' % ( lent,
                         'X', posAct+lengthLet, 'Y', 0, 'Z', down))))
            fileID.write(str(('%s %c%f %c%f %c%f\n' % ( rapide,
                         'X', posAct+lengthLet, 'Y', 0, 'Z', up))))
            posAct = posAct+lengthLet
    elif elem == 'L':
            fileID.write(str(('%s %c%f %c%f %c%f\n' % (
                         rapide, 'X', posAct, 'Y', 0, 'Z', up))))
            fileID.write(str(('%s %c%f %c%f %c%f\n' % (
                         lent, 'X', posAct, 'Y', 0, 'Z', down))))
            fileID.write(str(('%s %c%f %c%f %c%f\n' % ( lent,
                         'X', posAct, 'Y', hightLet, 'Z', down))))
            fileID.write(str(('%s %c%f %c%f %c%f\n' % (
                         rapide, 'X', posAct, 'Y', hightLet, 'Z', up))))
            fileID.write(str(('%s %c%f %c%f %c%f\n' % (
                         rapide, 'X', posAct, 'Y', 0, 'Z', up))))
            fileID.write(str(('%s %c%f %c%f %c%f\n' % (
                         lent, 'X', posAct, 'Y', 0, 'Z', down))))
            fileID.write(str(('%s %c%f %c%f %c%f\n' % ( lent,
                         'X', posAct+lengthLet, 'Y', 0, 'Z', down))))
            fileID.write(str(('%s %c%f %c%f %c%f\n' % ( rapide,
                         'X', posAct+lengthLet, 'Y', 0, 'Z', up))))
            posAct = posAct+lengthLet
    elif elem == 'M':
            fileID.write(str(('%s %c%f %c%f %c%f\n' % (
                         rapide, 'X', posAct, 'Y', 0, 'Z', up))))
            fileID.write(str(('%s %c%f %c%f %c%f\n' % (
                         lent, 'X', posAct, 'Y', 0, 'Z', down))))
            fileID.write(str(('%s %c%f %c%f %c%f\n' % ( lent,
                         'X', posAct, 'Y', hightLet, 'Z', down))))
            fileID.write(str(('%s %c%f %c%f %c%f\n' % ( lent, 'X',
                         posAct+lengthLet/2, 'Y', hightLet/2, 'Z', down))))
            fileID.write(str(('%s %c%f %c%f %c%f\n' % ( lent, 'X',
                         posAct+lengthLet, 'Y', hightLet, 'Z', down))))
            fileID.write(str(('%s %c%f %c%f %c%f\n' % ( lent,
                         'X', posAct+lengthLet, 'Y', 0, 'Z', down))))
            fileID.write(str(('%s %c%f %c%f %c%f\n' % ( rapide,
                         'X', posAct+lengthLet, 'Y', 0, 'Z', up))))
            posAct = posAct+lengthLet
    elif elem == 'N':
            fileID.write(str(('%s %c%f %c%f %c%f\n' % (
                         rapide, 'X', posAct, 'Y', 0, 'Z', up))))
            fileID.write(str(('%s %c%f %c%f %c%f\n' % (
                         lent, 'X', posAct, 'Y', 0, 'Z', down))))
            fileID.write(str(('%s %c%f %c%f %c%f\n' % ( lent,
                         'X', posAct, 'Y', hightLet, 'Z', down))))
            fileID.write(str(('%s %c%f %c%f %c%f\n' % ( lent,
                         'X', posAct+lengthLet, 'Y', 0, 'Z', down))))
            fileID.write(str(('%s %c%f %c%f %c%f\n' % ( lent, 'X',
                         posAct+lengthLet, 'Y', hightLet, 'Z', down))))
            fileID.write(str(('%s %c%f %c%f %c%f\n' % ( rapide,
                         'X', posAct+lengthLet, 'Y', hightLet, 'Z', up))))
            posAct = posAct+lengthLet
    elif elem == 'O':
            fileID.write(str(('%s %c%f %c%f %c%f\n' % ( rapide, 'X',
                         posAct+lengthLet, 'Y', hightLet*3/4, 'Z', up))))
            fileID.write(str(('%s %c%f %c%f %c%f\n' % ( lent, 'X',
                         posAct+lengthLet, 'Y', hightLet*3/4, 'Z', down))))
            fileID.write(str(('%s %c%f %c%f %c%f %c%f\n' % ( tourAntihoraire, 'X',
                         posAct+lengthLet-hightLet/4, 'Y', hightLet, 'I', -hightLet/4, 'J', 0))))
            fileID.write(str(('%s %c%f %c%f %c%f\n' % ( lent, 'X',
                         posAct+hightLet/4, 'Y', hightLet, 'Z', down))))
            fileID.write(str(('%s %c%f %c%f %c%f %c%f\n' % ( tourAntihoraire,
                         'X', posAct, 'Y', hightLet*3/4, 'I', 0, 'J', -hightLet/4))))
            fileID.write(str(('%s %c%f %c%f %c%f\n' % ( lent,
                         'X', posAct, 'Y', hightLet/4, 'Z', down))))
            fileID.write(str(('%s %c%f %c%f %c%f %c%f\n' % ( tourAntihoraire,
                         'X', posAct+hightLet/4, 'Y', 0, 'I', hightLet/4, 'J', 0))))
            fileID.write(str(('%s %c%f %c%f %c%f\n' % ( lent, 'X',
                         posAct+lengthLet-hightLet/4, 'Y', 0, 'Z', down))))
            fileID.write(str(('%s %c%f %c%f %c%f %c%f\n' % ( tourAntihoraire,
                         'X', posAct+lengthLet, 'Y', hightLet/4, 'I', 0, 'J', hightLet/4))))
            fileID.write(str(('%s %c%f %c%f %c%f\n' % ( lent, 'X',
                         posAct+lengthLet, 'Y', hightLet*3/4, 'Z', down))))
            fileID.write(str(('%s %c%f %c%f %c%f\n' % ( rapide, 'X',
                         posAct+lengthLet, 'Y', hightLet*3/4, 'Z', up))))
            posAct = posAct+lengthLet
    elif elem == 'P':
            fileID.write(str(('%s %c%f %c%f %c%f\n' % (
                         rapide, 'X', posAct, 'Y', 0, 'Z', up))))
            fileID.write(str(('%s %c%f %c%f %c%f\n' % (
                         lent, 'X', posAct, 'Y', 0, 'Z', down))))
            fileID.write(str(('%s %c%f %c%f %c%f\n' % ( lent,
                         'X', posAct, 'Y', hightLet, 'Z', down))))
            fileID.write(str(('%s %c%f %c%f %c%f\n' % ( lent, 'X',
                         posAct+lengthLet-hightLet/4, 'Y', hightLet, 'Z', down))))
            fileID.write(str(('%s %c%f %c%f %c%f %c%f\n' % ( tourHoraire, 'X',
                         posAct+lengthLet-hightLet/4, 'Y', hightLet/2, 'I', 0, 'J', -hightLet/4))))
            fileID.write(str(('%s %c%f %c%f %c%f\n' % ( lent,
                         'X', posAct, 'Y', hightLet/2, 'Z', down))))
            fileID.write(str(('%s %c%f %c%f %c%f\n' % ( rapide,
                         'X', posAct, 'Y', hightLet/2, 'Z', up))))
            posAct = posAct+lengthLet
    elif elem == 'Q':
            fileID.write(str(('%s %c%f %c%f %c%f\n' % ( rapide, 'X',
                         posAct+lengthLet, 'Y', hightLet*3/4, 'Z', up))))
            fileID.write(str(('%s %c%f %c%f %c%f\n' % ( lent, 'X',
                         posAct+lengthLet, 'Y', hightLet*3/4, 'Z', down))))
            fileID.write(str(('%s %c%f %c%f %c%f %c%f\n' % ( tourAntihoraire, 'X',
                         posAct+lengthLet-hightLet/4, 'Y', hightLet, 'I', -hightLet/4, 'J', 0))))
            fileID.write(str(('%s %c%f %c%f %c%f\n' % ( lent, 'X',
                         posAct+hightLet/4, 'Y', hightLet, 'Z', down))))
            fileID.write(str(('%s %c%f %c%f %c%f %c%f\n' % ( tourAntihoraire,
                         'X', posAct, 'Y', hightLet*3/4, 'I', 0, 'J', -hightLet/4))))
            fileID.write(str(('%s %c%f %c%f %c%f\n' % ( lent,
                         'X', posAct, 'Y', hightLet/4, 'Z', down))))
            fileID.write(str(('%s %c%f %c%f %c%f %c%f\n' % ( tourAntihoraire,
                         'X', posAct+hightLet/4, 'Y', 0, 'I', hightLet/4, 'J', 0))))
            fileID.write(str(('%s %c%f %c%f %c%f\n' % ( lent, 'X',
                         posAct+lengthLet-hightLet/4, 'Y', 0, 'Z', down))))
            fileID.write(str(('%s %c%f %c%f %c%f %c%f\n' % ( tourAntihoraire,
                         'X', posAct+lengthLet, 'Y', hightLet/4, 'I', 0, 'J', hightLet/4))))
            fileID.write(str(('%s %c%f %c%f %c%f\n' % ( lent, 'X',
                         posAct+lengthLet, 'Y', hightLet*3/4, 'Z', down))))
            fileID.write(str(('%s %c%f %c%f %c%f\n' % ( rapide, 'X',
                         posAct+lengthLet, 'Y', hightLet*3/4, 'Z', up))))
            fileID.write(str(('%s %c%f %c%f %c%f\n' % ( rapide, 'X',
                         posAct+lengthLet/2, 'Y', hightLet/2, 'Z', up))))
            fileID.write(str(('%s %c%f %c%f %c%f\n' % ( lent, 'X',
                         posAct+lengthLet/2, 'Y', hightLet/2, 'Z', down))))
            fileID.write(str(('%s %c%f %c%f %c%f\n' % ( lent,
                         'X', posAct+lengthLet, 'Y', 0, 'Z', down))))
            fileID.write(str(('%s %c%f %c%f %c%f\n' % ( rapide,
                         'X', posAct+lengthLet, 'Y', 0, 'Z', up))))
            posAct = posAct+lengthLet
    elif elem == 'R':
            fileID.write(str(('%s %c%f %c%f %c%f\n' % (
                         rapide, 'X', posAct, 'Y', 0, 'Z', up))))
            fileID.write(str(('%s %c%f %c%f %c%f\n' % (
                         lent, 'X', posAct, 'Y', 0, 'Z', down))))
            fileID.write(str(('%s %c%f %c%f %c%f\n' % ( lent,
                         'X', posAct, 'Y', hightLet, 'Z', down))))
            fileID.write(str(('%s %c%f %c%f %c%f\n' % ( lent, 'X',
                         posAct+lengthLet-hightLet/4, 'Y', hightLet, 'Z', down))))
            fileID.write(str(('%s %c%f %c%f %c%f %c%f\n' % ( tourHoraire, 'X',
                         posAct+lengthLet-hightLet/4, 'Y', hightLet/2, 'I', 0, 'J', -hightLet/4))))
            fileID.write(str(('%s %c%f %c%f %c%f\n' % ( lent,
                         'X', posAct, 'Y', hightLet/2, 'Z', down))))
            fileID.write(str(('%s %c%f %c%f %c%f\n' % ( lent,
                         'X', posAct+lengthLet, 'Y', 0, 'Z', down))))
            fileID.write(str(('%s %c%f %c%f %c%f\n' % ( rapide,
                         'X', posAct+lengthLet, 'Y', 0, 'Z', up))))
            posAct = posAct+lengthLet
    elif elem == 'S':
            fileID.write(str(('%s %c%f %c%f %c%f\n' % ( rapide, 'X',
                         posAct+lengthLet, 'Y', hightLet*3/4, 'Z', up))))
            fileID.write(str(('%s %c%f %c%f %c%f\n' % ( lent, 'X',
                         posAct+lengthLet, 'Y', hightLet*3/4, 'Z', down))))
            fileID.write(str(('%s %c%f %c%f %c%f %c%f\n' % ( tourAntihoraire, 'X',
                         posAct+lengthLet-hightLet/4, 'Y', hightLet, 'I', -hightLet/4, 'J', 0))))
            fileID.write(str(('%s %c%f %c%f %c%f\n' % ( lent, 'X',
                         posAct+hightLet/4, 'Y', hightLet, 'Z', down))))
            fileID.write(str(('%s %c%f %c%f %c%f %c%f\n' % ( tourAntihoraire,
                         'X', posAct+hightLet/4, 'Y', hightLet/2, 'I', 0, 'J', -hightLet/4))))
            fileID.write(str(('%s %c%f %c%f %c%f\n' % ( lent, 'X',
                         posAct+lengthLet-hightLet/4, 'Y', hightLet/2, 'Z', down))))
            fileID.write(str(('%s %c%f %c%f %c%f %c%f\n' % ( tourHoraire, 'X',
                         posAct+lengthLet-hightLet/4, 'Y', 0, 'I', 0, 'J', -hightLet/4))))
            fileID.write(str(('%s %c%f %c%f %c%f\n' % ( lent,
                         'X', posAct+hightLet/4, 'Y', 0, 'Z', down))))
            fileID.write(str(('%s %c%f %c%f %c%f %c%f\n' % ( tourHoraire,
                         'X', posAct, 'Y', hightLet/4, 'I', 0, 'J', hightLet/4))))
            fileID.write(str(('%s %c%f %c%f %c%f\n' % ( rapide,
                         'X', posAct, 'Y', hightLet/4, 'Z', up))))
            posAct = posAct+lengthLet
    elif elem == 'T':
            fileID.write(str(('%s %c%f %c%f %c%f\n' % ( rapide,
                         'X', posAct+lengthLet/2, 'Y', 0, 'Z', up))))
            fileID.write(str(('%s %c%f %c%f %c%f\n' % ( lent,
                         'X', posAct+lengthLet/2, 'Y', 0, 'Z', down))))
            fileID.write(str(('%s %c%f %c%f %c%f\n' % ( lent, 'X',
                         posAct+lengthLet/2, 'Y', hightLet, 'Z', down))))
            fileID.write(str(('%s %c%f %c%f %c%f\n' % ( rapide,
                         'X', posAct+lengthLet/2, 'Y', hightLet, 'Z', up))))
            fileID.write(str(('%s %c%f %c%f %c%f\n' % (
                         rapide, 'X', posAct, 'Y', hightLet, 'Z', up))))
            fileID.write(str(('%s %c%f %c%f %c%f\n' % ( lent,
                         'X', posAct, 'Y', hightLet, 'Z', down))))
            fileID.write(str(('%s %c%f %c%f %c%f\n' % ( lent, 'X',
                         posAct+lengthLet, 'Y', hightLet, 'Z', down))))
            fileID.write(str(('%s %c%f %c%f %c%f\n' % ( rapide,
                         'X', posAct+lengthLet, 'Y', hightLet, 'Z', up))))
            posAct = posAct+lengthLet
    elif elem == 'U':
            fileID.write(str(('%s %c%f %c%f %c%f\n' % (
                         rapide, 'X', posAct, 'Y', hightLet, 'Z', up))))
            fileID.write(str(('%s %c%f %c%f %c%f\n' % ( lent,
                         'X', posAct, 'Y', hightLet, 'Z', down))))
            fileID.write(str(('%s %c%f %c%f %c%f\n' % ( lent,
                         'X', posAct, 'Y', hightLet/4, 'Z', down))))
            fileID.write(str(('%s %c%f %c%f %c%f %c%f\n' % ( tourAntihoraire,
                         'X', posAct+hightLet/4, 'Y', 0, 'I', hightLet/4, 'J', 0))))
            fileID.write(str(('%s %c%f %c%f %c%f\n' % ( lent, 'X',
                         posAct+lengthLet-hightLet/4, 'Y', 0, 'Z', down))))
            fileID.write(str(('%s %c%f %c%f %c%f %c%f\n' % ( tourAntihoraire,
                         'X', posAct+lengthLet, 'Y', hightLet/4, 'I', 0, 'J', hightLet/4))))
            fileID.write(str(('%s %c%f %c%f %c%f\n' % ( lent, 'X',
                         posAct+lengthLet, 'Y', hightLet, 'Z', down))))
            fileID.write(str(('%s %c%f %c%f %c%f\n' % ( rapide,
                         'X', posAct+lengthLet, 'Y', hightLet, 'Z', up))))
            posAct = posAct+lengthLet
    elif elem == 'V':
            fileID.write(str(('%s %c%f %c%f %c%f\n' % (
                         rapide, 'X', posAct, 'Y', hightLet, 'Z', up))))
            fileID.write(str(('%s %c%f %c%f %c%f\n' % ( lent,
                         'X', posAct, 'Y', hightLet, 'Z', down))))
            fileID.write(str(('%s %c%f %c%f %c%f\n' % ( lent,
                         'X', posAct+lengthLet/2, 'Y', 0, 'Z', down))))
            fileID.write(str(('%s %c%f %c%f %c%f\n' % ( lent, 'X',
                         posAct+lengthLet, 'Y', hightLet, 'Z', down))))
            fileID.write(str(('%s %c%f %c%f %c%f\n' % ( rapide,
                         'X', posAct+lengthLet, 'Y', hightLet, 'Z', up))))
            posAct = posAct+lengthLet
    elif elem == 'W':
            fileID.write(str(('%s %c%f %c%f %c%f\n' % (
                         rapide, 'X', posAct, 'Y', hightLet, 'Z', up))))
            fileID.write(str(('%s %c%f %c%f %c%f\n' % ( lent,
                         'X', posAct, 'Y', hightLet, 'Z', down))))
            fileID.write(str(('%s %c%f %c%f %c%f\n' % ( lent,
                         'X', posAct+lengthLet/4, 'Y', 0, 'Z', down))))
            fileID.write(str(('%s %c%f %c%f %c%f\n' % ( lent, 'X',
                         posAct+lengthLet/2, 'Y', hightLet, 'Z', down))))
            fileID.write(str(('%s %c%f %c%f %c%f\n' % ( lent,
                         'X', posAct+lengthLet*3/4, 'Y', 0, 'Z', down))))
            fileID.write(str(('%s %c%f %c%f %c%f\n' % ( lent, 'X',
                         posAct+lengthLet, 'Y', hightLet, 'Z', down))))
            fileID.write(str(('%s %c%f %c%f %c%f\n' % ( rapide,
                         'X', posAct+lengthLet, 'Y', hightLet, 'Z', up))))
            posAct = posAct+lengthLet
    elif elem == 'X':
            fileID.write(str(('%s %c%f %c%f %c%f\n' % (
                         rapide, 'X', posAct, 'Y', hightLet, 'Z', up))))
            fileID.write(str(('%s %c%f %c%f %c%f\n' % ( lent,
                         'X', posAct, 'Y', hightLet, 'Z', down))))
            fileID.write(str(('%s %c%f %c%f %c%f\n' % ( lent,
                         'X', posAct+lengthLet, 'Y', 0, 'Z', down))))
            fileID.write(str(('%s %c%f %c%f %c%f\n' % ( rapide,
                         'X', posAct+lengthLet, 'Y', 0, 'Z', up))))
            fileID.write(str(('%s %c%f %c%f %c%f\n' % (
                         rapide, 'X', posAct, 'Y', 0, 'Z', up))))
            fileID.write(str(('%s %c%f %c%f %c%f\n' % (
                         lent, 'X', posAct, 'Y', 0, 'Z', down))))
            fileID.write(str(('%s %c%f %c%f %c%f\n' % ( lent, 'X',
                         posAct+lengthLet, 'Y', hightLet, 'Z', down))))
            fileID.write(str(('%s %c%f %c%f %c%f\n' % ( rapide,
                         'X', posAct+lengthLet, 'Y', hightLet, 'Z', up))))
            posAct = posAct+lengthLet
    elif elem == 'Y':
            fileID.write(str(('%s %c%f %c%f %c%f\n' % ( rapide,
                         'X', posAct+lengthLet/2, 'Y', 0, 'Z', up))))
            fileID.write(str(('%s %c%f %c%f %c%f\n' % ( lent,
                         'X', posAct+lengthLet/2, 'Y', 0, 'Z', down))))
            fileID.write(str(('%s %c%f %c%f %c%f\n' % ( lent, 'X',
                         posAct+lengthLet/2, 'Y', hightLet/2, 'Z', down))))
            fileID.write(str(('%s %c%f %c%f %c%f\n' % ( lent,
                         'X', posAct, 'Y', hightLet, 'Z', down))))
            fileID.write(str(('%s %c%f %c%f %c%f\n' % (
                         rapide, 'X', posAct, 'Y', hightLet, 'Z', up))))
            fileID.write(str(('%s %c%f %c%f %c%f\n' % ( rapide, 'X',
                         posAct+lengthLet/2, 'Y', hightLet/2, 'Z', up))))
            fileID.write(str(('%s %c%f %c%f %c%f\n' % ( lent, 'X',
                         posAct+lengthLet/2, 'Y', hightLet/2, 'Z', down))))
            fileID.write(str(('%s %c%f %c%f %c%f\n' % ( lent, 'X',
                         posAct+lengthLet, 'Y', hightLet, 'Z', down))))
            fileID.write(str(('%s %c%f %c%f %c%f\n' % ( rapide,
                         'X', posAct+lengthLet, 'Y', hightLet, 'Z', up))))
            posAct = posAct+lengthLet
    elif elem == 'Z':
            fileID.write(str(('%s %c%f %c%f %c%f\n' % ( rapide,
                         'X', posAct+lengthLet, 'Y', 0, 'Z', up))))
            fileID.write(str(('%s %c%f %c%f %c%f\n' % ( lent,
                         'X', posAct+lengthLet, 'Y', 0, 'Z', down))))
            fileID.write(str(('%s %c%f %c%f %c%f\n' % (
                         lent, 'X', posAct, 'Y', 0, 'Z', down))))
            fileID.write(str(('%s %c%f %c%f %c%f\n' % ( lent, 'X',
                         posAct+lengthLet, 'Y', hightLet, 'Z', down))))
            fileID.write(str(('%s %c%f %c%f %c%f\n' % ( lent,
                         'X', posAct, 'Y', hightLet, 'Z', down))))
            fileID.write(str(('%s %c%f %c%f %c%f\n' % (
                         rapide, 'X', posAct, 'Y', hightLet, 'Z', up))))
            posAct = posAct+lengthLet
    elif elem == '.':
            fileID.write(str(('%s %c%f %c%f %c%f\n' % (
                         rapide, 'X', posAct, 'Y', 0, 'Z', up))))
            fileID.write(str(('%s %c%f %c%f %c%f\n' % (
                         lent, 'X', posAct, 'Y', 0, 'Z', down))))
            fileID.write(str(('%s %c%f %c%f %c%f\n' % (
                         rapide, 'X', posAct, 'Y', 0, 'Z', up))))
    elif elem == ' ':
            posAct = posAct+lengthLet
posAct = posAct+space
#Write G-code to file
fileID.write(str(('%s %c%f %c%f %c%f\n' %(
             rapide, 'X', 0, 'Y', 0, 'Z', up))))

--- Python program Import G-Code ---
from os import path                   # Operating System API
from robolink import *      # RoboDK API
from robodk import *        # Robot toolbox

#Connect to RoboDK
RDK = Robolink()

# Get the robot by name:
robot = RDK.Item('M-6IB', 2)

#Set file directory for G-code file
filedirectory = path.expandvars(r'%USERPROFILE%\AppData\Local\Temp\letters.gcode')
#Set TCP_DrawingToolCorner as active tool
Drawing_tool = RDK.Item('TCP_DrawingToolCorner', 4)
robot.setPoseTool(Drawing_tool)

#Set Pencil_corner as active reference frame
Pencil_corner = RDK.Item('Pencil', 3)
robot.setPoseFrame(Pencil_corner)

#Create machining project
milling = RDK.AddMachiningProject('Millingsettings', robot)
#Set milling parameters
milling.setMachiningParameters(filedirectory,0,'NormalApproach=-50')
milling.setJoints([-46.931693, 64.148531, -65.163331, 39.068388, 105.370410, -198.556120]) # set the preferred start joints

--- program Final step (robot M-6IB) ---
  Call Attach_phone
  Set Ref.: End distination
  MoveJ (APP end )
  MoveL (End)
  Call Open gripper
  MoveL (APP end )

--- program Reset 2 (robot M-6IB) ---
  Replace objects

--- program Red phone assembly test (robot M-6IB) ---
  Set speed (200.0 mm/s)
  Call Assemble Red phone

--- program Blue phone assembly test (robot M-6IB) ---
  Set speed (200.0 mm/s)
  Call Assemble Blue phone

--- Python program Assemble red phone ---
# Type help("robolink") or help("robodk") for more information
# Press F5 to run the script
# Documentation: https://robodk.com/doc/en/RoboDK-API.html
# Reference:     https://robodk.com/doc/en/PythonAPI/index.html
# Note: It is not required to keep a copy of this file, your python script is saved with the station
from robolink import *    # RoboDK API
from robodk import *      # Robot toolbox
RDK = Robolink()
import time
# Notify user:
print('To edit this program:\nright click on the Python program, then, select "Edit Python script"')
text = 'ROBO'
# Program example:
item = RDK.Item('base')
gcodeGenerator = RDK.Item('Generate G-Code')
gcodeImport = RDK.Item('Import G-code')
assemble = RDK.Item('Assemble Red phone')

assemble.RunProgram()
while assemble.Busy():
    time.sleep(.300)
gcodeGenerator.RunProgram(['%s' % text])
while gcodeGenerator.Busy():
    time.sleep(.300)

gcodeImport.RunProgram()
while gcodeImport.Busy():
    time.sleep(.300)


Milling = RDK.Item('Millingsettings',8)
time.sleep(.300)
Milling.RunProgram()
while Milling.Busy():
    print('engraving..')
    time.sleep(.100)


Milling.Delete()
Milling = RDK.Item('Millingsettings')
Milling.Delete()


if item.Valid():
    print('Item selected: ' + item.Name())
    print('Item posistion: ' + repr(item.Pose()))

print('Items in the station:')
itemlist = RDK.ItemList()
print(itemlist)

--- program Reset (robot M-6IB) ---
  Replace objects
  Show objects

--- Python program Assemble blue phone ---
# Type help("robolink") or help("robodk") for more information
# Press F5 to run the script
# Documentation: https://robodk.com/doc/en/RoboDK-API.html
# Reference:     https://robodk.com/doc/en/PythonAPI/index.html
# Note: It is not required to keep a copy of this file, your python script is saved with the station
from robolink import *    # RoboDK API
from robodk import *      # Robot toolbox
RDK = Robolink()
import time
# Notify user:
print('To edit this program:\nright click on the Python program, then, select "Edit Python script"')

# Program example:
item = RDK.Item('base')
gcodeGenerator = RDK.Item('Generate G-Code')
gcodeImport = RDK.Item('Import G-code')
assemble = RDK.Item('Assemble Blue phone')

assemble.RunProgram()
while assemble.Busy():
    time.sleep(.300)

gcodeGenerator.RunProgram()
while gcodeGenerator.Busy():
    time.sleep(.300)

gcodeImport.RunProgram()
while gcodeImport.Busy():
    time.sleep(.300)


Milling = RDK.Item('Millingsettings',8)
time.sleep(.300)
Milling.RunProgram()
while Milling.Busy():
    print('engraving..')
    time.sleep(.300)


Milling.Delete()
Milling = RDK.Item('Millingsettings')
Milling.Delete()


if item.Valid():
    print('Item selected: ' + item.Name())
    print('Item posistion: ' + repr(item.Pose()))

print('Items in the station:')
itemlist = RDK.ItemList()
print(itemlist)

--- program AssembleInterior (robot M-6IB) ---
  Call Attach_PCB
  Call Detach_PCB
  Call Attach_Fuse
  Call Detach_Fuse1
  Call Attach_Fuse
  Call Detach_Fuse2
